(* Schneider Machine Expert - Basic project exercise_3.3, file version 2.9.0.0 *)
(* ProjectInformations: Name=Novo projeto *)

HARDWARE
  Cpu 0: TM221CE24R
  EthernetConfiguration: NetworkName=M221, IpAllocationMode=FixedAddress, IpAddress=0.0.0.0, SubnetMask=0.0.0.0
  SerialLineConfiguration: Baud=Baud19200, Parity=ParityEven, DataBits=DataBits8, StopBits=StopBits1, PhysicalMedium=PhysicalMediumRs485, TransmissionMode=TransmissionModeModbusRtu, SlaveId=1, Addressing=SlaveAddressing
  MastTask: UsePeriodScanMode=false, PeriodScan=100
  FastTask: Period=255
  CpuBehavior: StartingMode=StartAsPreviousState, AutoSaveRamOnEeprom=true, WatchdogPeriod=250

SYMBOLS  (address, symbol, comment, settings)
  %M0       SIG_IN_A_ATU
  %M1       SIG_IN_A_DESA
  %M2       SIG_IN_B_ATU
  %M3       SIG_IN_B_DESA
  %M4       SIG_T_A
  %M5       SIG_T_B
  %M6       SIG_OK
  %M20      SIG_LIGA_CONT_R
  %TM1      T_A  [Preset=3, Base=OneSecond]
  %TM2      T_B  [Preset=3, Base=OneSecond]
  %TM3      T_DESL  [Preset=3, Base=OneSecond]
  %I0.0     IN_A_ATU
  %I0.1     IN_A_DESA
  %I0.2     IN_B_ATU
  %I0.3     IN_B_DESA
  %Q0.1     OUT_CONT_R

POU Entradas
  (* SectionNumber=1 *)

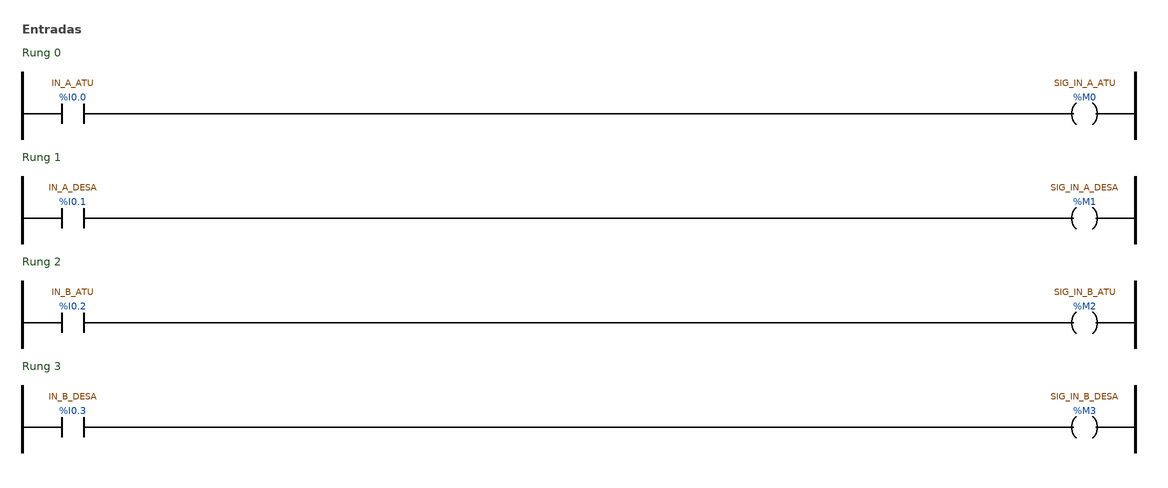

// Rung 0
  LD %I0.0                (* IN_A_ATU *)
  ST %M0                  (* SIG_IN_A_ATU *)
  // as ST:
  //   SIG_IN_A_ATU := IN_A_ATU;

// Rung 1
  LD %I0.1                (* IN_A_DESA *)
  ST %M1                  (* SIG_IN_A_DESA *)
  // as ST:
  //   SIG_IN_A_DESA := IN_A_DESA;

// Rung 2
  LD %I0.2                (* IN_B_ATU *)
  ST %M2                  (* SIG_IN_B_ATU *)
  // as ST:
  //   SIG_IN_B_ATU := IN_B_ATU;

// Rung 3
  LD %I0.3                (* IN_B_DESA *)
  ST %M3                  (* SIG_IN_B_DESA *)
  // as ST:
  //   SIG_IN_B_DESA := IN_B_DESA;

POU Lógicas
  (* SectionNumber=2 *)

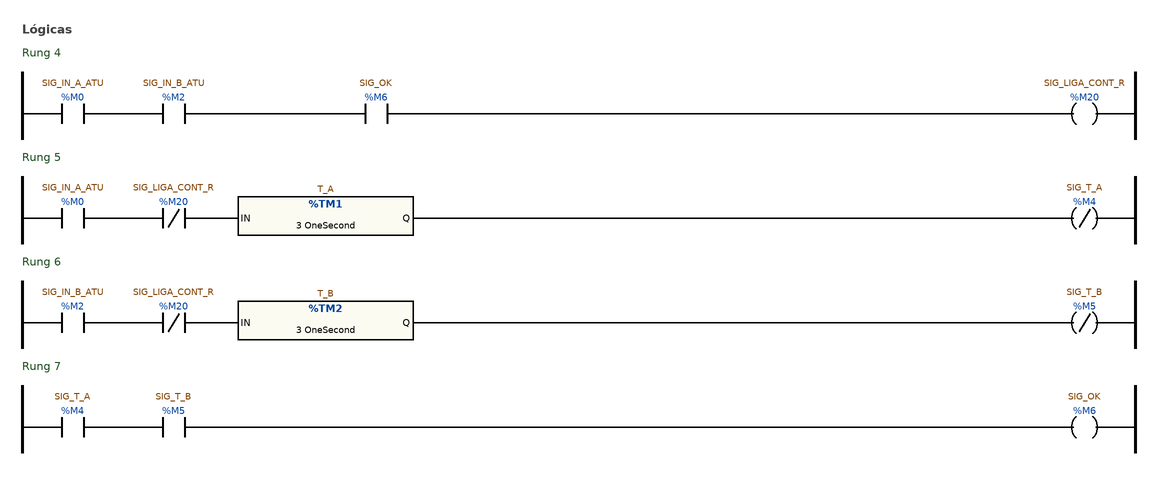

// Rung 4
  LD %M0                  (* SIG_IN_A_ATU *)
  AND %M2                 (* SIG_IN_B_ATU *)
  AND %M6                 (* SIG_OK *)
  ST %M20                 (* SIG_LIGA_CONT_R *)
  // as ST:
  //   SIG_LIGA_CONT_R := SIG_IN_A_ATU AND SIG_IN_B_ATU AND SIG_OK;

// Rung 5
  BLK %TM1                (* T_A *)
  LD %M0                  (* SIG_IN_A_ATU *)
  ANDN %M20               (* SIG_LIGA_CONT_R *)
  IN
  OUT_BLK
  LD Q
  STN %M4                 (* SIG_T_A *)
  END_BLK
  // as ST:
  //   T_A(IN := SIG_IN_A_ATU AND NOT SIG_LIGA_CONT_R);
  //   SIG_T_A := NOT T_A.Q;

// Rung 6
  BLK %TM2                (* T_B *)
  LD %M2                  (* SIG_IN_B_ATU *)
  ANDN %M20               (* SIG_LIGA_CONT_R *)
  IN
  OUT_BLK
  LD Q
  STN %M5                 (* SIG_T_B *)
  END_BLK
  // as ST:
  //   T_B(IN := SIG_IN_B_ATU AND NOT SIG_LIGA_CONT_R);
  //   SIG_T_B := NOT T_B.Q;

// Rung 7
  LD %M4                  (* SIG_T_A *)
  AND %M5                 (* SIG_T_B *)
  ST %M6                  (* SIG_OK *)
  // as ST:
  //   SIG_OK := SIG_T_A AND SIG_T_B;

POU Saídas
  (* SectionNumber=3 *)

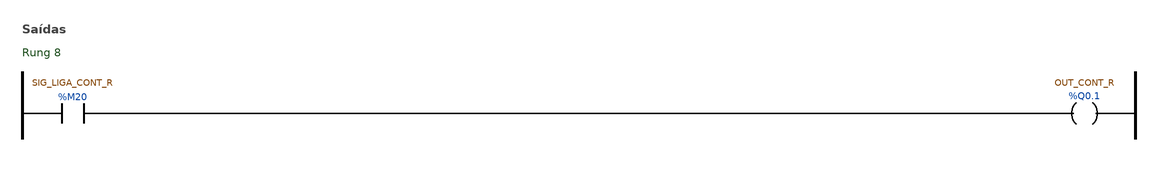

// Rung 8
  LD %M20                 (* SIG_LIGA_CONT_R *)
  ST %Q0.1                (* OUT_CONT_R *)
  // as ST:
  //   OUT_CONT_R := SIG_LIGA_CONT_R;
